TYPE MoverParameters_typ :
STRUCT
	
	Jerk			: LREAL;					// mm/s3
	Acceleration	: LREAL;					// mm/s2
	Deceleration	: LREAL;					// mm/s2
	Velocity		: LREAL;					// mm/s
	Direction		: Tc3_Mc3Definitions.MC_Direction;		// MC_Direction
	
END_STRUCT
END_TYPE

(* stored: Version 1.1.0.1, ProductVersion 3.1.4024.9
   DUT MoverParameters_typ: Id {bd3dfc46-8034-4584-b9a8-07f88efb1905} *)
